// Checks if string is boolean
FUNCTION F_ISBOOL : BOOL
VAR_INPUT
	sValue : T_Long_String;
END_VAR
VAR
END_VAR

F_TOUPPER(sValue);
F_ISBOOL := sValue = 'FALSE' OR_ELSE sValue = 'TRUE';

END_FUNCTION

(* stored: Version 1.1.0.1, ProductVersion 3.1.4024.4
   POU F_ISBOOL: Id {6e73a061-9665-4ba7-9d40-c4ac14cba95b}, SpecialFunc None *)
